INTERFACE IQualityInspection EXTENDS ZApplication.IUnit

END_INTERFACE

(* stored: Version 1.1.0.1
   Itf IQualityInspection: Id {8b9411ef-964d-42be-ae52-a1b9ecbc4f83} *)
